(* Logix 5000 project; controller programa vendor 1 type 14 code 151 rev 32.11; software revision 32.00 *)
// proyecto kit de control 18/07/2021

TASK MainTask (continuous, watchdog 500 ms) : MainProgram

MODULES
   Local : vendor 1 type 14 code 151 (Compact 0, rev 32.11)
      Analog_IO : Embedded (Compact 2, rev 1.1, Output RPI 80 ms)
      Counters : Embedded (Compact 3, rev 1.1, Output RPI 20 ms)
      Discrete_IO : Embedded (Compact 1, rev 3.1, Output RPI 20 ms)
END_MODULES

PROGRAM MainProgram   (* main routine MainRoutine *)
VAR
   salida0 : INT;
   salida1 : INT;
   salida2 : INT;
   salida3 : INT;
   salida4 : INT;
END_VAR

ROUTINE EntradasAnalogas   (* ladder *)
END_ROUTINE

ROUTINE EntradasDigitales   (* ladder *)
END_ROUTINE

ROUTINE MainRoutine   (* ladder *)
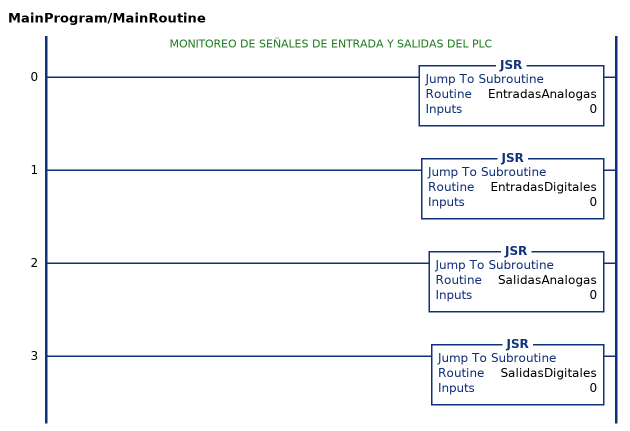
   // MONITOREO DE SEÑALES DE ENTRADA Y SALIDAS DEL PLC
   0: JSR(EntradasAnalogas,0);
   1: JSR(EntradasDigitales,0);
   2: JSR(SalidasAnalogas,0);
   3: JSR(SalidasDigitales,0);
END_ROUTINE

ROUTINE SalidasAnalogas   (* ladder *)
END_ROUTINE

ROUTINE SalidasDigitales   (* ladder *)
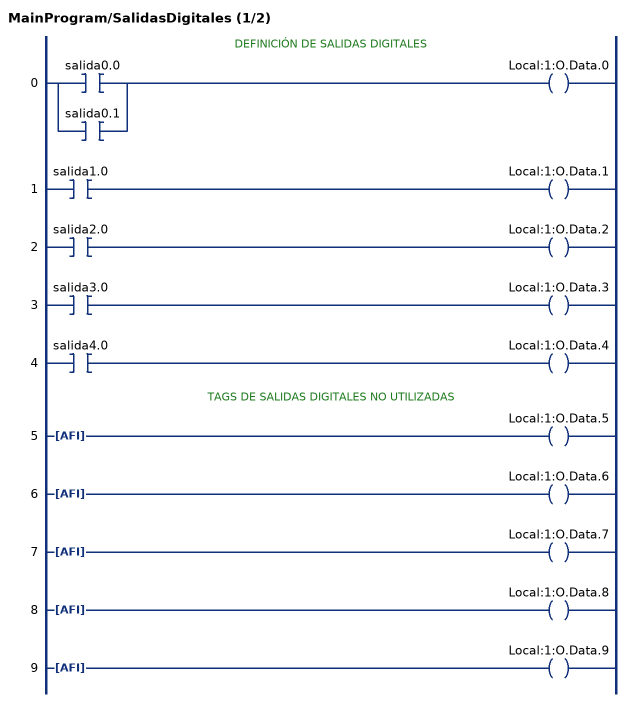
   // DEFINICIÓN DE SALIDAS DIGITALES
   0: [XIC(salida0.0) ,XIC(salida0.1) ]OTE(Local:1:O.Data.0);
   1: XIC(salida1.0)OTE(Local:1:O.Data.1);
   2: XIC(salida2.0)OTE(Local:1:O.Data.2);
   3: XIC(salida3.0)OTE(Local:1:O.Data.3);
   4: XIC(salida4.0)OTE(Local:1:O.Data.4);
   // TAGS DE SALIDAS DIGITALES NO UTILIZADAS
   5: AFI()OTE(Local:1:O.Data.5);
   6: AFI()OTE(Local:1:O.Data.6);
   7: AFI()OTE(Local:1:O.Data.7);
   8: AFI()OTE(Local:1:O.Data.8);
   9: AFI()OTE(Local:1:O.Data.9);
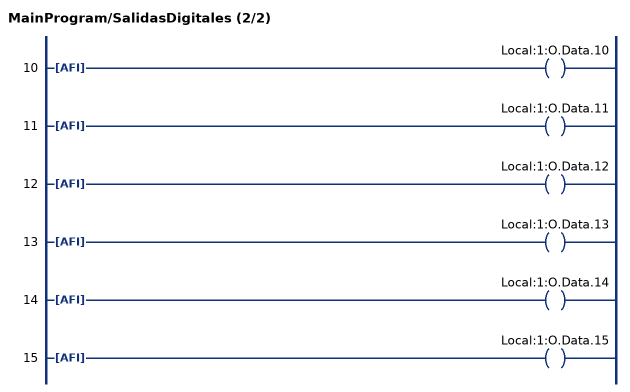
   10: AFI()OTE(Local:1:O.Data.10);
   11: AFI()OTE(Local:1:O.Data.11);
   12: AFI()OTE(Local:1:O.Data.12);
   13: AFI()OTE(Local:1:O.Data.13);
   14: AFI()OTE(Local:1:O.Data.14);
   15: AFI()OTE(Local:1:O.Data.15);
END_ROUTINE
END_PROGRAM
